FUNCTION_BLOCK ChangeDetect
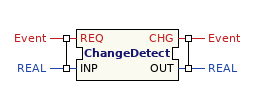
  EVENT_INPUT
    REQ WITH INP;
  END_EVENT
  EVENT_OUTPUT
    CHG WITH OUT;
  END_EVENT
  VAR_INPUT
    INP : REAL;
  END_VAR
  VAR_OUTPUT
    OUT : REAL;
  END_VAR
  VAR
    PREV : REAL := -1.0;
  END_VAR
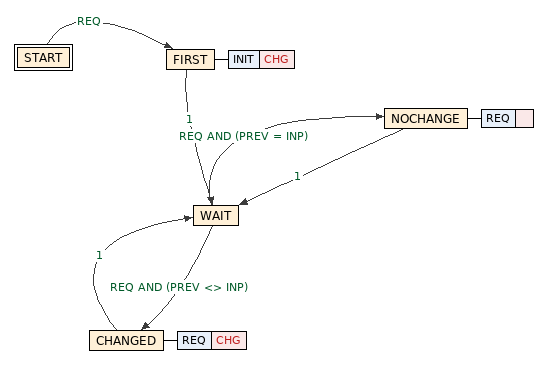
  EC_STATES
    START;
    NOCHANGE : REQ;
    CHANGED : REQ -> CHG;
    WAIT;
    FIRST : INIT -> CHG;
  END_STATES
  EC_TRANSITIONS
    WAIT TO NOCHANGE := REQ AND (PREV = INP);
    NOCHANGE TO WAIT := 1;
    WAIT TO CHANGED := REQ AND (PREV <> INP);
    CHANGED TO WAIT := 1;
    START TO FIRST := REQ;
    FIRST TO WAIT := 1;
  END_TRANSITIONS
  ALGORITHM INIT IN ST:
PREV := INP;
OUT := INP;
  END_ALGORITHM
  ALGORITHM REQ IN ST:
PREV := INP;
OUT := INP;
  END_ALGORITHM
END_FUNCTION_BLOCK
